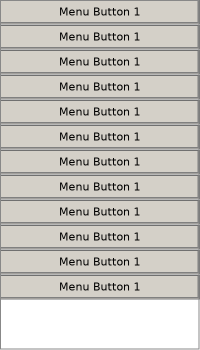
VISUALIZATION PopupMenu2  // 200x350
    Button (0,0 200x24), "Menu Button 1"
    Button (0,25 200x24), "Menu Button 1"
    Button (0,50 200x24), "Menu Button 1"
    Button (0,75 200x24), "Menu Button 1"
    Button (0,100 200x24), "Menu Button 1"
    Button (0,125 200x24), "Menu Button 1"
    Button (0,150 200x24), "Menu Button 1"
    Button (0,175 200x24), "Menu Button 1"
    Button (0,200 200x24), "Menu Button 1"
    Button (0,225 200x24), "Menu Button 1"
    Button (0,250 200x24), "Menu Button 1"
    Button (0,275 200x24), "Menu Button 1"
END_VISUALIZATION

(* stored: Version 1.1.0.1, ProductVersion 3.1.4024.11
   Visu PopupMenu2: Id {48d80a58-4c6e-0567-13a6-783e0d685fee} *)
